INTERFACE PUBLIC I_HeldCommands

METHOD PUBLIC Abort
END_METHOD

METHOD PUBLIC Stop
END_METHOD

METHOD PUBLIC Unhold
END_METHOD

END_INTERFACE

(* stored: Version 1.1.0.1, ProductVersion 3.1.4026.6
   Itf I_HeldCommands: Id {39048063-0d8e-08f0-155a-0e9a16743f7e}
   Method Abort: Id {97c2f5e3-ac64-4ebb-9359-7827843ff7c5}
   Method Stop: Id {a9c13afd-72fd-4d6c-b7b7-3fd0df820f6e}
   Method Unhold: Id {b1afe03d-1a2c-0ac6-15ac-16a5319470a8} *)
